// SIMATIC S7-200 project (STEP 7-Micro/WIN), CPU 224 REL 01.11

ORGANIZATION_BLOCK MAIN:OB1
TITLE=程序注释
// PLC通过PID算法自动调节加热器和冷却器的输出功率，确保反应釜温度稳定在200°C至220°C之间，满足化学反应的高效与安全需求。
// 系统在PLC首次上电时，调用子程序，设置PID循环定点为0.75（对应温度范围的75%）、PID循环增益为0.25、PID循环采样时间为0.1秒、PID积分时间为30分钟、PID微分时间为0.0（不启用微分控制）。
// 同时，系统将定时器间隔配置为100毫秒，并附加PID执行中断，保证PID控制以100毫秒的周期执行——只有这些参数正确初始化，系统才能正常运行。
BEGIN
Network 1 // // 次扫描时，调用初始化子例行程序

LD     SM0.1
CALL   SBR_0:SBR0
?000
END_ORGANIZATION_BLOCK

SUBROUTINE_BLOCK SBR_0:SBR0
TITLE=子例行程序注释
BEGIN
Network 1 // // 载入PID参数，并附加PID中断例行程序

// 网络注释
LD     SM0.0
MOVR   0.75, VD104           // 载入循环定点 = 注满75%
MOVR   0.25, VD112           // 载入循环增益 = 0.25
MOVR   0.1, VD116            // 载入循环采样时间 = 0.1秒
MOVR   30.0, VD120           // 载入积分时间 = 30分钟
MOVR   0.0, VD124            // 设置无微分计算
MOVB   100, SMB34            // 为定时中断INT_0
// 设置定时间隔（100毫秒）。
ATCH   INT_0:INT0, 10        // 设置定时中断，激活
// PID执行。
ENI                          // 启用中断
END_SUBROUTINE_BLOCK

INTERRUPT_BLOCK INT_0:INT0
TITLE=中断例行程序注释
BEGIN
Network 1 // 网络标题
// 网络注释
// 将PV标度为标准化实数
LD     SM0.0
ITD    AIW0, AC0             // 将整数数值转换为双整数
DTR    AC0, AC0              // 将双整数转换为实数
/R     32000.0, AC0          // 使数值正常化
MOVR   AC0, VD100            // 将正常化PV存储在循环表中
Network 2
//  位于自动模式时执行循环
// 
LD     I0.0
PID    VB100, 0
Network 3
//  将输出Mn标度为整数。
//  Mn是一个单极数值，不能为负数。
// 
LD     SM0.0
MOVR   VD108, AC0            // 将循环输出移至累加器
*R     32000.0, AC0          // 标度累加器中的数值
ROUND  AC0, AC0              // 将实数转换为双整数
DTI    AC0, AC0              // 将双整数转换为整数
MOVW   AC0, AQW0             // 将数值写入模拟输出
END_INTERRUPT_BLOCK
